PROGRAM myPressure
VAR
	iResinP : UINT;
	iAcetoneP : UINT;
	iGunMacsP AT %I* : UINT;
	myAir :INT;
END_VAR



//resin and MEK pump pressure


//acetone pump pressure


//itv for chopper (may add chopper to spindle on hmi interface to adjust the itv value


//gun mac pressure

END_PROGRAM

(* stored: Version 1.1.0.1, ProductVersion 3.1.4024.11
   POU myPressure: Id {7dc6c810-46ab-4bfa-96ec-40ac1944ad14}, SpecialFunc None *)
